KUKA KRL data list: ROBNAME.dat

&ACCESS RV
&PARAM TEMPLATE = C:\KRC\Roboter\Template\vorgabe
&PARAM EDITMASK = *
DEFDAT robname

GLOBAL ENUM E_PROPERTY_ROBNAME GET, SET
GLOBAL ENUM E_ROBOTNAME_TYPE TYPE_1, TYPE_2, UNKNOWN
GLOBAL STRUC ST_ROBOTNAME_TYPE E_ROBOT_TYPE eType INT iNumber
DECL ST_ROBOT_TYPE stRobot={eType #UNKNOWN,iNumber 0}

ENDDAT
